PROGRAM ADS
VAR
	fbAdsConnector : AdsConnector;
END_VAR

fbAdsConnector();
fbAdsConnector.Execute();

END_PROGRAM

(* stored: Version 1.1.0.1, ProductVersion 3.1.4024.0
   POU ADS: Id {42a8e07c-6d94-4347-bca1-6ed4d597561c}, SpecialFunc None *)
